Yaskawa INFORM job: ROS_R2.JBI

/JOB
//NAME ROS_R2
//POS
///NPOS 0,0,0,0,0,0
//INST
///DATE 2014/06/16 09:27
///ATTR SC,RW
///GROUP1 RB2
NOP
DOUT OT#(889) OFF
DOUT OT#(890) OFF
TIMER T=0.05
SKILLSND "ROS-START"
TSYNC 1
WAIT OT#(890)=ON
SKILLSND "ROS-STOP"
END
